ABB RAPID module: MainModule.mod

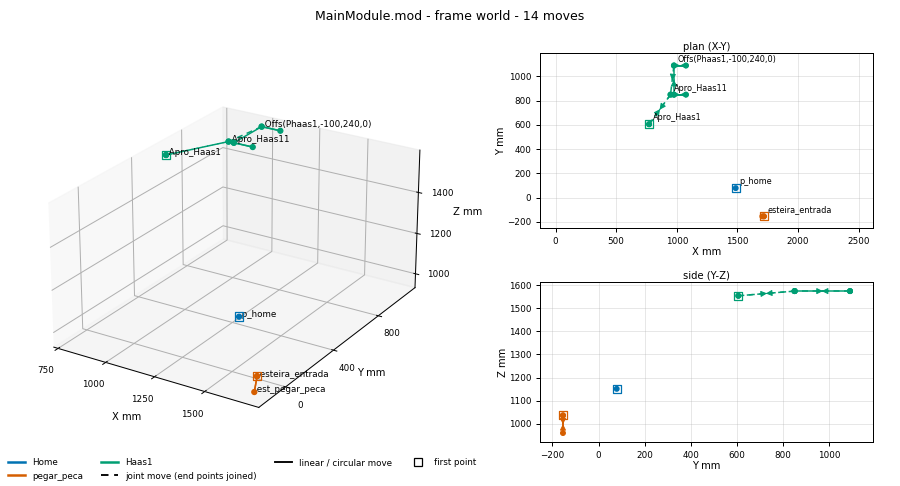
[picture p0: tool path of MainModule.mod in frame world, 14 of 14 moves have a stored position in this frame; points joined in program order, loops and branches not executed]
MODULE MainModule
	CONST robtarget esteira1:=[[474.32,-40.36,1231.00],[0.222911,0.184267,0.956969,-0.0237814],[-1,-1,0,0],[9E+09,9E+09,9E+09,9E+09,9E+09,9E+09]];
	CONST robtarget esteira11:=[[879.24,157.75,1277.21],[0.635608,0.0125581,0.761452,0.126631],[0,-1,0,1],[9E+09,9E+09,9E+09,9E+09,9E+09,9E+09]];
	CONST robtarget mov1:=[[474.31,300.61,1231.01],[0.222921,0.184246,0.956972,-0.0237729],[0,-1,0,0],[9E+09,9E+09,9E+09,9E+09,9E+09,9E+09]];
	CONST robtarget mov11:=[[232.90,300.63,1230.99],[0.222921,0.184229,0.956975,-0.0237824],[0,-1,0,0],[9E+09,9E+09,9E+09,9E+09,9E+09,9E+09]];
	CONST robtarget mov21:=[[423.12,160.14,1229.37],[0.195685,0.178528,0.964053,-0.020879],[0,-1,0,0],[9E+09,9E+09,9E+09,9E+09,9E+09,9E+09]];
	CONST robtarget mov31:=[[15.94,-538.00,1405.45],[0.15586,0.881367,0.378347,-0.236121],[-1,-1,0,0],[9E+09,9E+09,9E+09,9E+09,9E+09,9E+09]];
	CONST robtarget mov41:=[[122.33,-498.02,1606.31],[0.863559,0.224805,0.277511,-0.355972],[-1,-1,0,1],[9E+09,9E+09,9E+09,9E+09,9E+09,9E+09]];
	TASK PERS wobjdata mesa:=[FALSE,TRUE,"",[[1352.56,-126.662,1234.19],[0.989528,-0.00175601,-0.0022972,0.14431]],[[0,0,0],[1,0,0,0]]];
	TASK PERS wobjdata mesa2:=[FALSE,TRUE,"",[[1197.29,412.682,1233.04],[0.79976,-0.0015868,-0.000765591,-0.600317]],[[0,0,0],[1,0,0,0]]];
	CONST robtarget p_home:=[[1485.64,78.48,1150.93],[5.25263E-07,0.743875,0.668319,-3.07988E-07],[0,-1,1,0],[9E+09,9E+09,9E+09,9E+09,9E+09,9E+09]];
	CONST robtarget pRoX1:=[[201.28,328.12,163.98],[4.20989E-06,-0.101161,-0.99487,1.25289E-06],[0,-1,0,0],[9E+09,9E+09,9E+09,9E+09,9E+09,9E+09]];
	CONST robtarget pRoX11:=[[192.57,316.89,1.12],[4.91149E-05,-0.101174,-0.994869,8.7877E-06],[0,-1,0,0],[9E+09,9E+09,9E+09,9E+09,9E+09,9E+09]];
	CONST robtarget pInicial:=[[192.56,316.89,1.12],[4.97777E-05,-0.101174,-0.994869,8.76852E-06],[0,-1,0,0],[9E+09,9E+09,9E+09,9E+09,9E+09,9E+09]];
	CONST robtarget pInicial10:=[[192.56,316.89,1.10],[5.78358E-05,-0.101176,-0.994869,8.5355E-06],[0,-1,0,0],[9E+09,9E+09,9E+09,9E+09,9E+09,9E+09]];
	CONST robtarget pRoX21:=[[-149.70,325.88,339.59],[0.403996,0.190313,0.894633,0.0141371],[0,-1,0,0],[9E+09,9E+09,9E+09,9E+09,9E+09,9E+09]];
	VAR signaldo signaldo1;
	VAR bool flag1:=FALSE;
	TASK PERS tooldata caneta1:=[TRUE,[[-19.0299,12.9732,151.98],[0.0912258,-0.700157,0.0928062,0.702029]],[0.5,[0,0,0],[1,0,0,0],0,0,0]];
	TASK PERS tooldata Atuador:=[TRUE,[[-24.5396,-27.9623,140.131],[1,0,0,0]],[1,[-211,-56.9,311.4],[1,0,0,0],0,0,0.118]];
	CONST robtarget p_home10:=[[1712.85,-152.14,997.63],[0.0171986,0.801222,0.598101,0.00481647],[-1,-1,1,0],[9E+09,9E+09,9E+09,9E+09,9E+09,9E+09]];
	CONST robtarget p_home20:=[[1712.85,-152.13,997.63],[0.0171975,0.801221,0.598101,0.00481885],[-1,-1,1,0],[9E+09,9E+09,9E+09,9E+09,9E+09,9E+09]];
	CONST robtarget esteira_entrada:=[[1718.01,-154.28,1036.02],[0.0144755,0.801274,0.598115,0.00278515],[-1,-1,1,0],[9E+09,9E+09,9E+09,9E+09,9E+09,9E+09]];
	CONST robtarget esteira_entrada10:=[[1712.85,-152.14,997.63],[0.0171975,0.801222,0.598101,0.00481761],[-1,-1,1,0],[9E+09,9E+09,9E+09,9E+09,9E+09,9E+09]];
	CONST robtarget est_pegar_peca:=[[1704.96,-154.35,959.43],[0.014427,0.801282,0.598107,0.00271751],[-1,-1,1,0],[9E+09,9E+09,9E+09,9E+09,9E+09,9E+09]];
	CONST robtarget Apro_Haas1:=[[771.68,605.18,1553.97],[0.700122,0.0991232,0.700128,0.0991226],[0,-1,1,0],[9E+09,9E+09,9E+09,9E+09,9E+09,9E+09]];
	CONST robtarget Apro_Haas11:=[[948.20,849.12,1574.27],[0.716821,0.166241,0.674634,0.0583183],[0,-2,1,0],[9E+09,9E+09,9E+09,9E+09,9E+09,9E+09]];
	CONST robtarget Apro_Haas21:=[[1076.14,849.16,1574.27],[0.716822,0.166232,0.674634,0.0583291],[0,-2,1,0],[9E+09,9E+09,9E+09,9E+09,9E+09,9E+09]];
	CONST robtarget Phaas1:=[[1076.14,849.16,1574.27],[0.716822,0.166231,0.674635,0.0583262],[0,-2,1,0],[9E+09,9E+09,9E+09,9E+09,9E+09,9E+09]];
	CONST robtarget Apro_Haas31:=[[948.20,849.12,1574.27],[0.716821,0.166242,0.674633,0.0583159],[0,-2,1,0],[9E+09,9E+09,9E+09,9E+09,9E+09,9E+09]];
	PROC main()
		<SMT>
	ENDPROC
	PROC Home()
		MoveJ p_home, v1000, z50, tool0;
	ENDPROC
	PROC pegar_peca()
		MoveJ esteira_entrada, v1000, fine, Atuador;
		MoveL est_pegar_peca, v1000, fine, Atuador;
		Set DO_10_atuador;
		WaitTime 3;
		MoveL esteira_entrada, v1000, z50, Atuador;
	ENDPROC
	PROC Haas1()
		MoveJ Apro_Haas1, v1000, z50, Atuador;
		MoveJ Apro_Haas11, v1000, z50, Atuador;
		MoveL Offs(Phaas1,-100,0,0), v1000, z50, Atuador;
		MoveL Phaas1, v100, fine, Atuador;
		MoveL Offs(Phaas1,-100,0,0), v1000, z50, Atuador;
		MoveL Offs(Phaas1,-100,240,0), v1000, z50, Atuador;
		MoveL Offs(Phaas1,0,240,0), v1000, z50, Atuador;
		MoveL Offs(Phaas1,-100,240,0), v1000, z50, Atuador;
		MoveJ Apro_Haas11, v1000, z50, Atuador;
		MoveJ Apro_Haas1, v1000, z50, Atuador;
	ENDPROC
ENDMODULE
